FUNCTION_BLOCK FB_ValveCommandFactory
VAR
END_VAR

METHOD CreateCommand : I_Command
VAR_INPUT
	valve : I_Valve;
	target : E_ValvePosition;
	description : STRING;
END_VAR
VAR	
	point : POINTER TO FB_ValveMoveCommand;
END_VAR
point := __NEW(FB_ValveMoveCommand(valve := valve, target := target, description := description));
CreateCommand := point^;
END_METHOD

END_FUNCTION_BLOCK

(* stored: Version 1.1.0.1
   POU FB_ValveCommandFactory: Id {acd8081e-3e38-4701-9b8d-5e428312f198}, SpecialFunc None
   Method CreateCommand: Id {f2c53adb-7a58-464d-9c22-7893029afccc} *)
